INTERFACE I_MotionAxisNC EXTENDS I_MotionAxisCommon

PROPERTY LimBwdEnable : BOOL
GET
END_GET
SET
END_SET
END_PROPERTY

PROPERTY LimFwdEnable : BOOL
GET
END_GET
SET
END_SET
END_PROPERTY

PROPERTY LimHome : BOOL
GET
END_GET
SET
END_SET
END_PROPERTY

END_INTERFACE

(* stored: Version 1.1.0.1
   Itf I_MotionAxisNC: Id {988e1537-42fa-4f3b-9835-b781579a345f}
   Property LimBwdEnable: Id {9b524dc8-ec6b-43f0-b711-98e44add3824}
   Get Get: Id {08bd27e3-9813-40a8-97d1-fba2b5b94922}
   Set Set: Id {008cffef-5d72-4f01-bef9-dfa538a736c1}
   Property LimFwdEnable: Id {8701f4da-08d0-4f0c-97c2-7f7351b1ff2a}
   Get Get: Id {ff1dea93-3860-43be-a364-014c90fd8ed5}
   Set Set: Id {885f42ff-aa99-470c-a0b1-41b648319e83}
   Property LimHome: Id {91a731c7-16ed-42dd-a83a-6787494f1a7f}
   Get Get: Id {6e46de07-f8a9-4f92-98f3-95a9910c688c}
   Set Set: Id {fa7195f6-f66e-4eea-a1f2-9d4ea8913f5d} *)
